PROGRAM MAIN
VAR
END_VAR

END_PROGRAM

(* stored: Version 1.1.0.1
   POU MAIN: Id {df389ca3-de85-4c10-9bab-104593257845} *)
